TYPE ST_AssemblyOutputs :
STRUCT
    clamp : ST_CylinderOutputs;
    press : ST_CylinderOutputs;
    ejector : ST_CylinderOutputs;
END_STRUCT
END_TYPE

(* stored: Version 1.1.0.1
   DUT ST_AssemblyOutputs: Id {2770e69a-bac2-45a1-a1a6-90d9d2701a71} *)
